INTERFACE I_ControlBox

METHOD Mode
VAR_INPUT
END_VAR
END_METHOD

END_INTERFACE

(* stored: Version 1.1.0.1, ProductVersion 3.1.4024.12
   Itf I_ControlBox: Id {9f885559-3305-4675-809f-2cf4e90fe19b}
   Method Mode: Id {c5c82611-b5c0-4eb8-9171-b21927bf4a1d} *)
